(* CODESYS project LS Electric.library
   Author: Ziga Javornik
   Version: 0.0.1.1
   Description: LS Electric device libraries collection.
   Title: ZigaLibs.LsElectric
   Placeholder: ZigaLibs.LsElectric
   DefaultNamespace: ZigaLibs.LsElectric
   Company: Ziga Javornik

Project tree, tasks and I/O mapping:
  libraries: Tc2_Standard, * (Beckhoff Automation GmbH); Tc2_System, * (Beckhoff Automation GmbH); Tc3_Module, * (Beckhoff Automation GmbH); TcUnit, 1.3.1 (www.tcunit.org); ZigaLibs.Core, * (Ziga Javornik); ZigaLibs.Logging, * (Ziga Javornik)
  GVLs/
  SOURCE/
    L7NHA/
      DUTs/
        CoE/
          data type ST_L7NHA_CoE
        data type E_L7NHA_DriveState
        data type E_L7NHA_ErrorId
        data type E_L7NHA_HomingMethod
        data type E_L7NHA_ModeOfOperation
        data type ST_L7NHA_DataFromDrive
        data type ST_L7NHA_DataToDrive
        data type ST_L7NHA_DigitalInputs
        data type ST_L7NHA_EthercatData
        data type ST_L7NHA_GearRatio
        data type ST_L7NHA_HomingCommands
        data type ST_L7NHA_HomingStatus
        data type ST_L7NHA_MotionFeedback
        data type ST_L7NHA_PositioningCommands
        data type ST_L7NHA_PositioningStatus
        data type ST_L7NHA_ProfileTorqueCommands
        data type ST_L7NHA_UserUnitParams
        data type ST_L7NHA_VelocityCommands
      function block FB_L7NHA [ST]: SetGearRatio, SetHomingMethod, DisableVoltage, EnableOperation, FaultReset, Halt, Shutdown, SwitchOn, SwitchOnEnableOperation, Homing, ProfilePosition, ProfileTorque, ProfileVelocity, CalculateTorque, FB_init, GetDriveState
  TESTS/
    Test suites/
      function block FB_SUT_Tests [ST]: TestXX_Template
    program PRG_TESTS [ST]
*)

// SOURCE/L7NHA/DUTs/CoE/ST_L7NHA_CoE
TYPE ST_L7NHA_CoE :
STRUCT
	HomingMethod	: ZigaLibs_Core.ST_CoeEntry_SINT := (Index := 16#6098);
	GearRatio_Motor	: ZigaLibs_Core.ST_CoeEntry_DINT := (Index := 16#6091, Subindex := 1);
	GearRatio_Shaft	: ZigaLibs_Core.ST_CoeEntry_DINT := (Index := 16#6091, Subindex := 2);
END_STRUCT
END_TYPE

// SOURCE/L7NHA/DUTs/E_L7NHA_DriveState
{attribute 'qualified_only'}
{attribute 'strict'}
{attribute 'to_string'}
// Drive states based on the CiA402 state machine
TYPE E_L7NHA_DriveState :
(
	SWITCH_ON_DISABLED,
	READY_TO_SWITCH_ON,
	SWITCHED_ON,
	OPERATION_ENABLED,
	QUICK_STOP_ACTIVE,
	FAULT_REACTION_ACTIVE,
	FAULT
);
END_TYPE

// SOURCE/L7NHA/DUTs/E_L7NHA_ErrorId
{attribute 'qualified_only'}
{attribute 'to_string'}
// Drive error ID - same as the error displayed on the servo 7SEG display
TYPE E_L7NHA_ErrorId :
(
	NO_ERROR := 0,
	IPM_FAULT := 16#10,
	IPM_TEMPERATURE := 16#11,
	OVER_CURRENT := 16#14,
	CURRENT_OFFSET := 16#15,
	CURRENT_LIMIT_EXCEEDED := 16#16,
	CONTINIOUS_OVERLOAD := 16#21,
	DRIVE_TEMPERATURE_1 := 16#22,
	REGENERATION_OVERLOAD := 16#23,
	MOTOR_CABLE_OPEN := 16#24,
	SURROUNDING_TEMPERATURE := 16#25,
	ENCODER_TEMPERATURE := 16#26,
	ECONDER_COMMUNICATION := 16#30,
	ENCODER_CABLE_OPEN := 16#31,
	ENCODER_DATA := 16#32,
	MOTOR_SETTINGS := 16#33,
	Z_PHASE_OPEN := 16#34,
	LOW_BATTERY := 16#35,
	SINUSODIAL_ENCODER_AMPLITUDE := 16#36,
	SINUSODIAL_ENCODER_FREQUENCY := 16#37,
	ENCODER_SETTING_ERROR := 16#38,
	UNDER_VOLTAGE := 16#40,
	OVER_VOLTAGE := 16#41,
	MAIN_POWER_FAIL := 16#42,
	CONTROL_POWER_FAIL := 16#43,
	OVER_SPEED_LIMIT := 16#50,
	POS_FOLLOWING := 16#51,
	EXCESSIVE_SPEED_DEVIATION := 16#53,
	PARAMETER_CHECKSUM := 16#63,
	FACTORY_SETTING := 16#71
) UINT;
END_TYPE

// SOURCE/L7NHA/DUTs/E_L7NHA_HomingMethod
{attribute 'qualified_only'}
{attribute 'strict'}
{attribute 'to_string'}
// All the different homing methods
TYPE E_L7NHA_HomingMethod :
(
	DISABLED 									:= 0,	// Homing is disabled
	NEGATIVE_SWITCH_INDEX_REVERSE_DIRECTION 	:= 1, 	// The drive returns to the home position with the negative limit switch (NOT) and the Index (Z) pulse while driving in the reverse direction.
	POSITIVE_SWITCH_INDEX_FORWARD_DIRECTION 	:= 2, 	// The drive returns to the home position with the positive limit switch (POT) and the Index (Z) pulse while driving in the forward direction.
	HOME_SWITCH_INDEX_FORWARD_DIRECTION_7 		:= 7,	// The drive returns to the home position with the home switch (HOME) and the Index (Z) pulse while driving in the forward direction. When the positive limit switch (POT) is input during homing, the drive will switch its driving direction.
	HOME_SWITCH_INDEX_FORWARD_DIRECTION_8 		:= 8,	// The drive returns to the home position with the home switch (HOME) and the Index (Z) pulse while driving in the forward direction. When the positive limit switch (POT) is input during homing, the drive will switch its driving direction.
	HOME_SWITCH_INDEX_FORWARD_DIRECTION_9 		:= 9,	// The drive returns to the home position with the home switch (HOME) and the Index (Z) pulse while driving in the forward direction. When the positive limit switch (POT) is input during homing, the drive will switch its driving direction.
	HOME_SWITCH_INDEX_FORWARD_DIRECTION_10 		:= 10,	// The drive returns to the home position with the home switch (HOME) and the Index (Z) pulse while driving in the forward direction. When the positive limit switch (POT) is input during homing, the drive will switch its driving direction.
	HOME_SWITCH_INDEX_REVERSE_DIRECTION_11 		:= 11,	// The drive returns to the home position with the home switch (HOME) and the Index (Z) pulse while driving in the reverse direction. When the negative limit switch (NOT) is input during homing, the drive will switch its driving direction.
	HOME_SWITCH_INDEX_REVERSE_DIRECTION_12 		:= 12,	// The drive returns to the home position with the home switch (HOME) and the Index (Z) pulse while driving in the reverse direction. When the negative limit switch (NOT) is input during homing, the drive will switch its driving direction.
	HOME_SWITCH_INDEX_REVERSE_DIRECTION_13 		:= 13,	// The drive returns to the home position with the home switch (HOME) and the Index (Z) pulse while driving in the reverse direction. When the negative limit switch (NOT) is input during homing, the drive will switch its driving direction.
	HOME_SWITCH_INDEX_REVERSE_DIRECTION_14 		:= 14,	// The drive returns to the home position with the home switch (HOME) and the Index (Z) pulse while driving in the reverse direction. When the negative limit switch (NOT) is input during homing, the drive will switch its driving direction.
	HOME_SWITCH_FORWARD_DIRECTION 				:= 24,	// The drive returns to the home position with the home switch (HOME) while driving in the forward direction. When the positive limit switch (POT) is input during homing, the drive will switch its driving direction.
	HOME_SWITCH_REVERSE_DIRECTION 				:= 28,	// The drive returns to the home position with the home switch (HOME) while driving in the reverse direction. When the negative limit switch (NOT) is input during homing, the drive will switch its driving direction.
	INDEX_REVERSE_DIRECTION 					:= 33,	// The drive returns to the home position with the Index (Z) pulse while driving in the reverse direction.
	INDEX_FORWARD_DIRECTION 					:= 34,	// The drive returns to the home position with the Index (Z) pulse while driving in the forward direction.
	TO_THE_CURRENT_POSITION 					:= 35,	// Sets the current position as the origin.
	NEGATIVE_STOPPER_INDEX_REVERSE_DURECTION	:= -1,	// The drive returns to the home position with the negative stopper and the Index (Z) pulse while driving in the reverse direction.
	POSITIVE_STOPPER_INDEX_FORWARD_DIRECTION 	:= -2,	// The drive returns to the home position with the positive stopper and the Index (Z) pulse while driving in the forward direction.
	REVERSE_STOPPER_REVERSE_DIRECTION 			:= -3,	// The drive returns to the home position with the negative stopper while driving in the reverse direction.
	POSITIVE_STOPPER_FORWARD_DIRECTION 			:= -4	// The drive returns to the home position with the positive stopper while driving in the forward direction.
) SINT;
END_TYPE

// SOURCE/L7NHA/DUTs/E_L7NHA_ModeOfOperation
{attribute 'qualified_only'}
{attribute 'to_string'}
// All the possible drive modes
TYPE E_L7NHA_ModeOfOperation :
(
	PROFILE_POSITION 		:= 1,
	PROFILE_VELOCITY 		:= 3,
	PROFILE_TORQUE 			:= 4,
	HOMING					:= 6,
	INTERPOLATED_POSITION	:= 7,
	CYCLIC_SYNC_POSITION	:= 8,
	CYCLIC_SYNC_VELOCITY	:= 9,
	CYCLIC_SYNC_TORQUE		:= 10
)SINT;
END_TYPE

// SOURCE/L7NHA/DUTs/ST_L7NHA_DataFromDrive
TYPE ST_L7NHA_DataFromDrive :
STRUCT
	StatusWord			: WORD;		// Status word
	ModeOfOperation		: SINT;		// Actual mode of operation
	ErrorCode			: E_L7NHA_ErrorId;		// Most recent error code
	DigitalInputs		: UDINT;	// Info on various digital inputs
	MotionFeedback		: ST_L7NHA_MotionFeedback;	// Motion feedback from the drive
END_STRUCT
END_TYPE

// SOURCE/L7NHA/DUTs/ST_L7NHA_DataToDrive
TYPE ST_L7NHA_DataToDrive :
STRUCT
	// Control
	ControlWord					: WORD;	// Control word
	ModeOfOperation				: SINT;	// Mode of operation
	
	// Positioning mode
	ProfileVelocity				: DINT;	// Target velocity in PP mode
	TargetPosition				: DINT;	// Target position in PP mode
	MaximumProfileVelocity		: UDINT; // Maximum velocity in PP mode
	ProfileAcceleration			: UDINT; // Deceleration UU/s^2 when using PP mode
	ProfileDeceleration			: UDINT; // Acceleration UU/s^2 when using PP mode
	
	TorqueCommands	: ST_L7NHA_ProfileTorqueCommands;
	
	// Velocity mode
	TargetVelocity				: DINT;	// Target velocity in PV mode
END_STRUCT
END_TYPE

// SOURCE/L7NHA/DUTs/ST_L7NHA_DigitalInputs
TYPE ST_L7NHA_DigitalInputs :
STRUCT
	POT_SW		: BOOL;
	NOT_SW		: BOOL;
	HOME_SW		: BOOL;
	DI1_OPEN	: BOOL;
	DI2_OPEN	: BOOL;
	DI3_OPEN	: BOOL;
	DI4_OPEN	: BOOL;
	DI5_OPEN	: BOOL;
	DI6_OPEN	: BOOL;
	DI7_OPEN	: BOOL;
	DI8_OPEN	: BOOL;
	STO_OPEN	: BOOL;
END_STRUCT
END_TYPE

// SOURCE/L7NHA/DUTs/ST_L7NHA_EthercatData
TYPE ST_L7NHA_EthercatData :
STRUCT
	MasterNetID		: AMSNETID;
	SlaveAddress	: UINT;
END_STRUCT
END_TYPE

// SOURCE/L7NHA/DUTs/ST_L7NHA_GearRatio
TYPE ST_L7NHA_GearRatio :
STRUCT
	Motor	: DINT;
	Shaft	: DINT;
END_STRUCT
END_TYPE

// SOURCE/L7NHA/DUTs/ST_L7NHA_HomingCommands
TYPE ST_L7NHA_HomingCommands :
STRUCT
	Start							: BOOL;	// Starts homing procedure
	Enable							: BOOL;	// Homing will only be execute if this flag is set to true
	HomingMethod					: E_L7NHA_HomingMethod; // Defines homing method that will be used for the axis - bEnableCoeReadWrite needs to be set to TRUE for this parameter to be written
	Acceleration					: UDINT; // Acceleration in UU/s^2 - bEnableCoeReadWrite needs to be set to TRUE for this parameter to be written
	SpeedWhileSearchingForSwitch	: UDINT; // Speed at which homing will be moving axis when searching for the physical switch - bEnableCoeReadWrite needs to be set to TRUE for this parameter to be written
	SpeedWhileSearchingForZero		: UDINT; // Speed at which homing will be moving axis after switch has been found and axis is looking for index pulse - bEnableCoeReadWrite needs to be set to TRUE for this parameter to be written
END_STRUCT
END_TYPE

// SOURCE/L7NHA/DUTs/ST_L7NHA_HomingStatus
TYPE ST_L7NHA_HomingStatus :
STRUCT
	InProgress			: BOOL; // Homing in progress
	NotStarted			: BOOL; // Homing stopped or not started
	TargetNotReached	: BOOL; // Performed homing operation, but the not reach the target
	Completed			: BOOL; // Homing completed
	ErrorSpeedNotZero	: BOOL; // Homing error; speed not equal to 0
	ErrorSpeedIsZero	: BOOL; // Homing error; speed equal to 0
END_STRUCT
END_TYPE

// SOURCE/L7NHA/DUTs/ST_L7NHA_MotionFeedback
TYPE ST_L7NHA_MotionFeedback :
STRUCT
	TargetTorque		: INT;	// Target torque in .1 * rated torque
	ActualTorque		: INT;	// Torque .1 * rated torque
	
	TargetPosition		: DINT;	// Target position in user units
	ActualPosition		: DINT;	// Position in user units

	TargetMotorSpeed	: INT;	
	ActualMotorSpeed	: INT;	// Motor speed in RPM

	TargetVelocity		: DINT;	// Target velocity in user units
	ActualVelocity		: DINT;	// Velocity in user units
END_STRUCT
END_TYPE

// SOURCE/L7NHA/DUTs/ST_L7NHA_PositioningCommands
TYPE ST_L7NHA_PositioningCommands :
STRUCT
	VelocitySetpoint		: DINT;		// Velocity setpoint when in positioning mode
	MaxVelocity				: UDINT;	// Maximum allowed velocity when in positioning mode
	TargetPosition			: DINT;		// Target position
	GoToPosition			: BOOL;		// Positioning will be executed on rising edge
	ImmediatePositioning	: BOOL;		// If set to TRUE target position will be sent to the drive immediately and executed - otherwise the target only updates on GoToPosition call	
	EnablePositioning		: BOOL;		// Positioning will only be executed when this flag is set to true
END_STRUCT
END_TYPE

// SOURCE/L7NHA/DUTs/ST_L7NHA_PositioningStatus
TYPE ST_L7NHA_PositioningStatus :
STRUCT
	TargetPositionReached	 		: BOOL;	// TRUE if position has been reached
	SetpointAcknowledged			: BOOL;	// TRUE if new setpoint has been acknowledged
	PositionalError					: BOOL;	// TRUE if positioning error is detected
END_STRUCT
END_TYPE

// SOURCE/L7NHA/DUTs/ST_L7NHA_ProfileTorqueCommands
TYPE ST_L7NHA_ProfileTorqueCommands :
STRUCT
	TargetTorque			: UINT; // Target value - 0.1% of rated torque
	MaxTorque				: UINT; // Limits torque in both directions - 0.1% of rated torque
	MaximumProfileVelocity 	: UDINT; // Maximum velocity when driving using the torque mode - UU/s
	TorqueSlope				: UDINT; // Slope of the generated torque profile - 0.1%/s
	PositiveTorqueLimit		: UINT;	// Limit when driving in positive direction - 0.1%
	NegativeTorqueLimit		: UINT;	// Limit when driving in negative direction - 0.1%
	TorqueOffset			: UINT;	// Offset added to the TargeTorque
END_STRUCT
END_TYPE

// SOURCE/L7NHA/DUTs/ST_L7NHA_UserUnitParams
// Specifies custom user unit data that can be used for further conversion from within the block
TYPE ST_L7NHA_UserUnitParams :
STRUCT
	(* Use this to specify if you want to use custom user unit, different from the one set on the drive. 
	This can be useful if you have low user unit and want to sue higher unit inside the program since 
	scaling is done within the block for simplciyt sake. If you don't want to use actual units leave this at 1 (or 0 - internal check will ommit any calculation if set to 0).
	Example:
		- Gearbox ratio is set so that user unit is 1um.
		- You want to use milimeters as your unit inside the program.
		- Set the divisor to 1000 - UU outside the block is then 1mm = 1value, instead of 1000 = 1000um = 1mm..*)
	GearboxRatioUnitDivisor	: DINT := 1;
	
	(*User unit for velocity is by deafult in UU/s. Use this to automatically convert velocity to UU/<CustomVelocityTimeUnitDivisor>*seconds
	Example:
		- You have set up the gearbox to be in milimeters per 1 unit.
		- You want the speed to be in mm/minute instead of defautl mm/second.
		- Set this parameter to 60, this way velocity feedback will be multiplied by 60, which will return velocity in mm/min 
		  and velocity setpoint will be divided by 60 to specify the speed to the drive in UU/seconds, which is the only option.*)	
	CustomVelocityTimeUnitDivisor		: REAL := 1;
END_STRUCT
END_TYPE

// SOURCE/L7NHA/DUTs/ST_L7NHA_VelocityCommands
TYPE ST_L7NHA_VelocityCommands :
STRUCT
	VelocitySetpoint	: DINT;	// Target velocity in UU/s used in Profile Velocity mode
END_STRUCT
END_TYPE

// SOURCE/L7NHA/FB_L7NHA
FUNCTION_BLOCK FB_L7NHA EXTENDS ZigaLibs_Core.FB_HasInstanceNameAndPath

VAR_INPUT
	bEnable					: BOOL;	// Enable axis
	bReset					: BOOL;	// Reset if an eror is present
	bHalt					: BOOL; // Halts current operation - after setting this to FALSE previous operation is continuoued
	bQuickStop				: BOOL;	// Drive will execute a quick stop
	
	nAcceleration			: UDINT;	// Axis acceleration in UU/s^2
	nDeceleration			: UDINT;	// Axis deceleration in UU/s^
	
	eModeOfOperation		: E_L7NHA_ModeOfOperation;	// Mode of operation
	
	stVelocityCommands		: ST_L7NHA_VelocityCommands;		// Velocity commands when in profile velocity mode
	stPositioningCommands	: ST_L7NHA_PositioningCommands;		// Positioning commands when in profile position mode
	stHomingCommands		: ST_L7NHA_HomingCommands;			// Homing commands when in homing sequence
	stProfileTorqueCommands	: ST_L7NHA_ProfileTorqueCommands;	// Profile torque commands when using Profile Torque mode
	
	fRatedTorque			: REAL; // Rated torque in mNm - required for torque calculation

	stGearRatio				: ST_L7NHA_GearRatio;	// Used to set gear ratio
END_VAR

VAR_OUTPUT
	eAxisState			: E_L7NHA_DriveState;	// Axis state, actual state reported back from drive
	
	eErrorCode			: E_L7NHA_ErrorId;	// Error code, if drive is in fault state
	
	bHomingRequired		: BOOL;	// If homing is required, this flag will be set to true (usually after a power reset)
	
	bMovingPositive		: BOOL;	// Indicating axis is rotating in positive direction
	bMovingNegative		: BOOL;	// Indicating axis is rotating in negative direction
	
	stPositioningStatus	: ST_L7NHA_PositioningStatus;	// Status of the positioning procedure - only valid when in positioning mode
	stHomingStatus		: ST_L7NHA_HomingStatus;		// Status of the homing procedure - only valid when in homing mode
	
	fCalculatedActualTorque	: REAL;
	fCalculatedTargetTorque	: REAL;
	
	eActualModeOfOperation	: E_L7NHA_ModeOfOperation;
	stMotionFeedback		: ST_L7NHA_MotionFeedback;	// Motion feedback from the drive

	stDigitalInputs	:		 ST_L7NHA_DigitalInputs;
	
	bModeOfOperationNotImplemented	: BOOL;	// Will be TRUE if the selected mode of operation is not implemented (axis has to be in enabled state for this flag to be valid!)
END_VAR

// Local variables
VAR
	eAxisStateInternal					: E_L7NHA_DriveState;
	stDataToDriveInternal				: ST_L7NHA_DataToDrive;
	TonCommandTimeout					: Tc2_Standard.TON := (PT := T#1S);
	RtrigMoveToPosition					: Tc2_Standard.R_TRIG;
	RtrigStartHoming					: Tc2_Standard.R_TRIG;
	nPreviousPosition					: DINT;
	RtrigResetTrigger					: Tc2_Standard.R_TRIG;
	RtrigHomingFinished					: Tc2_Standard.R_TRIG;
	TonMotorMovingStatusValid			: Tc2_Standard.TON;
	RtrigModeOfOperationNotImplemented	: Tc2_Standard.R_TRIG;
	eModeOfOpereationOld				: E_L7NHA_ModeOfOperation;
	_logger								: REFERENCE TO ZigaLibs_Logging.I_Logger;
	_sb									: ZigaLibs_Core.FB_StringBuilder;
	_coeEntries							: ST_L7NHA_CoE;
END_VAR

// IO
VAR
	stDataFromDrive	AT %I* : ST_L7NHA_DataFromDrive;
	stDataToDrive	AT %Q* : ST_L7NHA_DataToDrive;
	stAmsAddress	AT %I* : Global.AMSADDR;
END_VAR

// Sometimes axis wont go to enabled - in that case a timeout should be triggered
TonCommandTimeout(in := eAxisStateInternal = E_L7NHA_DriveState.OPERATION_ENABLED);
// Reset triggering
RtrigResetTrigger(CLK := bReset);


// Abs encoder value is not valid if bit 14 is FALSE (homing has not been completed yet after a power reset/encoder error)
bHomingRequired := stDataFromDrive.StatusWord.14 = FALSE;

// Calling halt will overwrite this - to enable automatic clearing, setting it to false by default
stDataToDriveInternal.ControlWord.8 := FALSE;

// State machine based on the drive's feedback
eAxisStateInternal := THIS^.GetDriveState();

bModeOfOperationNotImplemented := FALSE;
		
// State machine based on actual state reported back from the drive
CASE eAxisStateInternal OF
	E_L7NHA_DriveState.SWITCH_ON_DISABLED:	
		IF bEnable THEN
			Shutdown();
		ELSE
			DisableVoltage();
		END_IF
	
	E_L7NHA_DriveState.READY_TO_SWITCH_ON:
		IF NOT TonCommandTimeout.Q THEN
			SwitchOnEnableOperation();
		END_IF
		
	E_L7NHA_DriveState.OPERATION_ENABLED:
		TonCommandTimeout.IN := FALSE;
		SwitchOnEnableOperation();

		// Execute different mode based on mode of operation setting
		CASE eModeOfOperation OF
			E_L7NHA_ModeOfOperation.PROFILE_POSITION:
				ProfilePosition();
				
			E_L7NHA_ModeOfOperation.PROFILE_VELOCITY:
				ProfileVelocity();
				
			E_L7NHA_ModeOfOperation.HOMING:
				Homing();
				
			E_L7NHA_ModeOfOperation.PROFILE_TORQUE:
				ProfileTorque();
				
			ELSE
				bModeOfOperationNotImplemented := TRUE;
				IF eModeOfOperation <> eModeOfOpereationOld THEN
					IF __ISVALIDREF(_logger) THEN
						_logger.LogError(_sb.Reset()
							.AddString('L7NHA axis ')
							.AddWithDblQuotationMarks(THIS^.InstanceName)
							.AddString(': Mode of operation is not supported! Selected mode is ')
							.AddWithDblQuotationMarks(TO_STRING(eModeOfOperation))
							.Create());
					END_IF
				END_IF
		END_CASE
		
	E_L7NHA_DriveState.FAULT:
		IF RtrigResetTrigger.Q THEN
			FaultReset();
		ELSE
			stDataToDriveInternal.ControlWord.7 := FALSE;
		END_IF

END_CASE

// Override any command if enable is false (transitioning states) - exception is fault, where reset needs to be sent
IF NOT bEnable AND eAxisStateInternal <> E_L7NHA_DriveState.FAULT THEN
	DisableVoltage();
END_IF

// Halt - has a different meaning in PP,PV or homing 
// Usally it "pauses" the current procedure and after halt is set to FALSE drive will proceed where it left off
IF bHalt THEN
	Halt();
END_IF

// Quick stop
IF bQuickStop THEN
	stDataToDriveInternal.ControlWord.1 := bQuickStop;
	stDataToDriveInternal.ControlWord.2 := NOT bQuickStop;
END_IF

// Setting acceleration/deceleration always
stDataToDriveInternal.ProfileAcceleration := nAcceleration;
stDataToDriveInternal.ProfileDeceleration := nDeceleration;

// Mode of operation
stDataToDriveInternal.ModeOfOperation := eModeOfOperation;


// =======================================================================
// ==================== SETTING FB OUTPUTS ===============================
// =======================================================================

// Axis state
eAxisState := eAxisStateInternal;

// Overwriting status for positioning/homing if not in that mode
// Clear homing status if not in that mode
IF eModeOfOperation <> E_L7NHA_ModeOfOperation.HOMING THEN
	MEMSET(
		destAddr := ADR(stHomingStatus),
		n := SIZEOF(stHomingStatus),
		fillByte := 0);
END_IF
 
// Clear positioning status if not in that mode
IF eModeOfOperation <> E_L7NHA_ModeOfOperation.PROFILE_POSITION THEN
	MEMSET(
		destAddr := ADR(stPositioningStatus),
		n := SIZEOF(stPositioningStatus),
		fillByte := 0);
END_IF

// Motion status
TonMotorMovingStatusValid(
	IN := nPreviousPosition <> stDataFromDrive.MotionFeedback.ActualPosition,
	PT := T#30MS);

bMovingPositive := (nPreviousPosition < stDataFromDrive.MotionFeedback.ActualPosition) AND TonMotorMovingStatusValid.Q;
bMovingNegative := (nPreviousPosition > stDataFromDrive.MotionFeedback.ActualPosition) AND TonMotorMovingStatusValid.Q;
nPreviousPosition := stDataFromDrive.MotionFeedback.ActualPosition;

// Digital inputs mapping
stDigitalInputs.NOT_SW := stDataFromDrive.DigitalInputs.0;
stDigitalInputs.POT_SW := stDataFromDrive.DigitalInputs.1;
stDigitalInputs.DI1_OPEN := stDataFromDrive.DigitalInputs.16;
stDigitalInputs.DI2_OPEN := stDataFromDrive.DigitalInputs.17;
stDigitalInputs.DI3_OPEN := stDataFromDrive.DigitalInputs.18;
stDigitalInputs.DI4_OPEN := stDataFromDrive.DigitalInputs.19;
stDigitalInputs.DI5_OPEN := stDataFromDrive.DigitalInputs.20;
stDigitalInputs.DI6_OPEN := stDataFromDrive.DigitalInputs.21;
stDigitalInputs.DI7_OPEN := stDataFromDrive.DigitalInputs.22;
stDigitalInputs.DI8_OPEN := stDataFromDrive.DigitalInputs.23;
stDigitalInputs.STO_OPEN := stDataFromDrive.DigitalInputs.31;

// Error code
IF eErrorCode <> stDataFromDrive.ErrorCode THEN
	IF __ISVALIDREF(_logger) THEN
		IF stDataFromDrive.ErrorCode = E_L7NHA_ErrorId.NO_ERROR THEN
			_logger.LogInfo(_sb.Reset()
				.AddString('L7NHA axis ')
				.AddWithDblQuotationMarks(THIS^.InstanceName)
				.AddString(' error no longer active.')
				.Create());
		ELSE
			_logger.LogError(_sb.Reset()
				.AddString('L7NHA axis ')
				.AddWithDblQuotationMarks(THIS^.InstanceName)
				.AddString(' error active! Error code: ')
				.AddString(TO_STRING(stDataFromDrive.ErrorCode))
				.AddString(' !')
				.Create());
		END_IF
	END_IF
END_IF

eErrorCode := stDataFromDrive.ErrorCode;

// Motion feedback from drive
stMotionFeedback := stDataFromDrive.MotionFeedback;
// Convert position/velocity to custom units

stMotionFeedback := stDataFromDrive.MotionFeedback;

fCalculatedActualTorque := CalculateTorque(fRatedTorque := fRatedTorque, nDriveTorqueFeedback := stDataFromDrive.MotionFeedback.ActualTorque);
fCalculatedTargetTorque := CalculateTorque(fRatedTorque := fRatedTorque, nDriveTorqueFeedback := stDataFromDrive.MotionFeedback.TargetTorque);

// Actual mode of operation, read from the drive
eActualModeOfOperation := stDataFromDrive.ModeOfOperation;

eModeOfOpereationOld := eModeOfOperation;

// =======================================================================
// ==================== SETTING OUTPUT STRUCTURE TO DRIVE ================
// =======================================================================
stDataToDrive := stDataToDriveInternal;

// Observes the stGearRatio.Shaft and stGearRatio.Motor. If the setting changes the new value is written to the CoE parameter.
METHOD pubLIC SetGearRatio : BOOL

VAR_INST
	coeReadWrite	: ZigaLibs_Core.FB_CoeReadWrite;
	sb				: ZigaLibs_Core.FB_StringBuilder;
	writeShaftDone 	: BOOL;
	writeMotorDone	: BOOL;
END_VAR
IF writeMotorDone = FALSE THEN
	IF coeReadWrite.WriteAny(
		Value := stGearRatio.Motor, 
		CoeEntry := ADR(_coeEntries.GearRatio_Motor), 
		SlaveAddr := stAmsAddress)
	THEN
		writeMotorDone := TRUE;
		IF __ISVALIDREF(_logger) then
			sb.Reset()
				.AddString('L7NHA axis ')
				.AddWithDblQuotationMarks(THIS^.InstanceName)
				.AddString(': Motor gear ratio changed to ')
				.AddString(TO_STRING(stGearRatio.Motor));
			_logger.LogInfo(sb.Create());
		END_IF
	END_IF	
END_IF

IF writeMotorDone THEN
	IF coeReadWrite.WriteAny(
		Value := stGearRatio.Shaft, 
		CoeEntry := ADR(_coeEntries.GearRatio_Motor), 
		SlaveAddr := stAmsAddress)
	THEN
		SetGearRatio := TRUE;
		writeMotorDone := FALSE;
		IF __ISVALIDREF(_logger) then
			sb.Reset()
				.AddString('L7NHA axis ')
				.AddWithDblQuotationMarks(THIS^.InstanceName)
				.AddString(': Shaft gear ratio changed to ')
				.AddString(TO_STRING(stGearRatio.Shaft));
			_logger.LogInfo(sb.Create());
		END_IF
	END_IF		
END_IF
END_METHOD

// Writes the current homing method provided in stHomingCommands.HomingMethod to the CoE of the axis. Returns TRUE when done
METHOD PUBLIC SetHomingMethod : BOOL
VAR_INST
	coeReadWrite	: ZigaLibs_Core.FB_CoeReadWrite;
	sb				: ZigaLibs_Core.FB_StringBuilder;
END_VAR
IF coeReadWrite.WriteAny(
		Value := stHomingCommands.HomingMethod, 
		CoeEntry := ADR(_coeEntries.HomingMethod), 
		SlaveAddr := stAmsAddress)
THEN 
	IF __ISVALIDREF(_logger) then
		sb.Reset()
			.AddString('L7NHA axis ')
			.AddWithDblQuotationMarks(THIS^.InstanceName)
			.AddString(': Homing method changing to ')
			.AddString(TO_STRING(stHomingCommands.HomingMethod));
		_logger.LogInfo(sb.Create());
	END_IF
	SetHomingMethod := TRUE;
END_IF
END_METHOD

METHOD PRIVATE DisableVoltage
stDataToDriveInternal.controlWord := 0;
END_METHOD

METHOD PRIVATE EnableOperation
stDataToDriveInternal.controlWord.0 := 0;
stDataToDriveInternal.controlWord.1 := 1;
stDataToDriveInternal.controlWord.2 := 1;
stDataToDriveInternal.controlWord.3 := 0;
stDataToDriveInternal.controlWord.4 := 0;
stDataToDriveInternal.controlWord.5 := 0;
stDataToDriveInternal.controlWord.6 := 0;
stDataToDriveInternal.controlWord.7 := 0;
END_METHOD

METHOD PRIVATE FaultReset
IF stDataToDriveInternal.controlWord.7 = 0 THEN
	stDataToDriveInternal.controlWord.7 := 1;
	stDataToDriveInternal.controlWord.0 := 0;
	stDataToDriveInternal.controlWord.1 := 0;
	stDataToDriveInternal.controlWord.2 := 0;
	stDataToDriveInternal.controlWord.3 := 0;
END_IF
END_METHOD

// Halts the axis for as long as called
METHOD PRIVATE Halt : BOOL
VAR_INPUT
END_VAR
stDataToDriveInternal.ControlWord.8 := TRUE;
END_METHOD

METHOD PRIVATE Shutdown
stDataToDriveInternal.controlWord.0 := 0;
stDataToDriveInternal.controlWord.1 := 1;
stDataToDriveInternal.controlWord.2 := 1;
stDataToDriveInternal.controlWord.7 := 0;
END_METHOD

METHOD PRIVATE SwitchOn
stDataToDriveInternal.controlWord.0 := 1;
stDataToDriveInternal.controlWord.1 := 1;
stDataToDriveInternal.controlWord.2 := 1;
stDataToDriveInternal.controlWord.3 := 0;
END_METHOD

METHOD PRIVATE SwitchOnEnableOperation
stDataToDriveInternal.controlWord.0 := 1;
stDataToDriveInternal.controlWord.1 := 1;
stDataToDriveInternal.controlWord.2 := 1;
stDataToDriveInternal.controlWord.3 := 1;
END_METHOD

ACTION Homing:
// Set the status of homing

// Hooming is in progress
stHomingStatus.InProgress := 
stDataFromDrive.StatusWord.10 = FALSE AND
stDataFromDrive.StatusWord.12 = FALSE AND
stDataFromDrive.StatusWord.13 = FALSE;

// Homing is not started
stHomingStatus.NotStarted := 
stDataFromDrive.StatusWord.10 = TRUE AND
stDataFromDrive.StatusWord.12 = FALSE AND
stDataFromDrive.StatusWord.13 = FALSE;	

// Target not reached	
stHomingStatus.TargetNotReached := 
stDataFromDrive.StatusWord.10 = FALSE AND
stDataFromDrive.StatusWord.12 = TRUE AND
stDataFromDrive.StatusWord.13 = FALSE;

// Homing completed
stHomingStatus.Completed := 
stDataFromDrive.StatusWord.10 = TRUE AND
stDataFromDrive.StatusWord.12 = TRUE AND
stDataFromDrive.StatusWord.13 = FALSE;

// Error - speed is not zero ????
stHomingStatus.ErrorSpeedNotZero := 
stDataFromDrive.StatusWord.10 = FALSE AND
stDataFromDrive.StatusWord.12 = FALSE AND
stDataFromDrive.StatusWord.13 = TRUE;

// Error - speed is zero ????
stHomingStatus.ErrorSpeedIsZero := 
stDataFromDrive.StatusWord.10 = TRUE AND
stDataFromDrive.StatusWord.12 = FALSE AND
stDataFromDrive.StatusWord.13 = TRUE;


RtrigStartHoming(CLK := stHomingCommands.Start);	
IF stHomingCommands.Enable = FALSE THEN
	stDataToDriveInternal.ControlWord.4 := FALSE;
ELSIF RtrigStartHoming.Q THEN
	stDataToDriveInternal.ControlWord.4 := TRUE;
END_IF

RtrigHomingFinished(CLK := stHomingStatus.Completed);
IF RtrigHomingFinished.Q THEN
	stDataToDriveInternal.ControlWord.4 := FALSE;
END_IF
END_ACTION

ACTION ProfilePosition:
// Positioning is only allowed if homing has been executed
IF NOT bHomingRequired THEN					
	// Set maximum velocity
	stDataToDriveInternal.MaximumProfileVelocity := stPositioningCommands.MaxVelocity;
	
	// Update target immediately - bit 5 is TRUE
	stDataToDriveInternal.ControlWord.5 := TRUE;
	
	// Trigger immediate update of setpoint by toggling the bit
	IF stPositioningCommands.EnablePositioning THEN
		// Toggling of bit 4 will execute the changes as soon as they are written
		IF stPositioningCommands.ImmediatePositioning THEN
			stDataToDriveInternal.ControlWord.4 := NOT stDataToDriveInternal.ControlWord.4;
			stDataToDriveInternal.ProfileVelocity := stPositioningCommands.VelocitySetpoint;
			stDataToDriveInternal.TargetPosition := stPositioningCommands.TargetPosition;
		ELSE
			// Bit 4 is only set for 1 cycle when requested by the GoToPosition trigger
			stDataToDriveInternal.ControlWord.4 := FALSE;
			// Sending values only on triger of GoToPosition property
			RtrigMoveToPosition(CLK := stPositioningCommands.GoToPosition);
			IF RtrigMoveToPosition.Q THEN
				stDataToDriveInternal.ControlWord.4 := TRUE;
				stDataToDriveInternal.ProfileVelocity := stPositioningCommands.VelocitySetpoint;
				stDataToDriveInternal.TargetPosition := stPositioningCommands.TargetPosition;
			END_IF
		END_IF
	ELSE
		Halt();
	END_IF
	
	// Positioning status from drive
	stPositioningStatus.TargetPositionReached := stDataFromDrive.StatusWord.10;
	stPositioningStatus.SetpointAcknowledged := stDataFromDrive.StatusWord.12;
	stPositioningStatus.PositionalError := stDataFromDrive.StatusWord.13;
ELSE
	// If homing has not been executed, halt axis
	Halt();
END_IF
END_ACTION

ACTION ProfileTorque:
stDataToDriveInternal.TorqueCommands := stProfileTorqueCommands;
END_ACTION

ACTION ProfileVelocity:
// Velocity mode is very simple - just send out the speed setpoint
stDataToDriveInternal.TargetVelocity := stVelocityCommands.VelocitySetpoint;
END_ACTION

METHOD PRIVATE CalculateTorque : REAL
VAR_INPUT
	fRatedTorque 			: REAL; // Rated torque in mNm
	nDriveTorqueFeedback 	: INT;	// Drives feedback (0.1% increments, -100%...+100%)
END_VAR
CalculateTorque := fRatedTorque * TO_REAL(nDriveTorqueFeedback);
END_METHOD

METHOD FB_init : BOOL
VAR_INPUT
	bInitRetains : BOOL; // if TRUE, the retain variables are initialized (warm start / cold start)
	bInCopyCode : BOOL;  // if TRUE, the instance afterwards gets moved into the copy code (online change)
	logger		: REFERENCE TO ZigaLibs_Logging.I_Logger; // If you do not want logging, simply set this variable to 0, internal checks will ommit any logging.		
END_VAR
_logger REF= logger;
END_METHOD

// Converts status word to a readable drive state enum
METHOD PRIVATE GetDriveState : E_L7NHA_DriveState
//================ SWITCH_ON_DISABLED =====================
IF stDataFromDrive.StatusWord.0 = FALSE AND
    stDataFromDrive.StatusWord.1 = FALSE AND
    stDataFromDrive.StatusWord.2 = FALSE AND
    stDataFromDrive.StatusWord.3 = FALSE AND
    stDataFromDrive.StatusWord.5 = TRUE AND 
    stDataFromDrive.StatusWord.6 = TRUE
THEN
	GetDriveState := E_L7NHA_DriveState.SWITCH_ON_DISABLED;

//================ READY_TO_SWITCH_ON =====================	
ELSIF stDataFromDrive.StatusWord.0 = TRUE AND
   	   stDataFromDrive.StatusWord.1 = FALSE AND
       stDataFromDrive.StatusWord.2 = FALSE AND
       stDataFromDrive.StatusWord.3 = FALSE AND
       stDataFromDrive.StatusWord.5 = TRUE AND 
       stDataFromDrive.StatusWord.6 = FALSE
THEN
	GetDriveState := E_L7NHA_DriveState.READY_TO_SWITCH_ON;	

//================ SWITCHED_ON ==========================	
ELSIF stDataFromDrive.StatusWord.0 = TRUE AND
   	   stDataFromDrive.StatusWord.1 = TRUE AND
       stDataFromDrive.StatusWord.2 = FALSE AND
       stDataFromDrive.StatusWord.3 = FALSE AND
       stDataFromDrive.StatusWord.5 = TRUE AND 
       stDataFromDrive.StatusWord.6 = FALSE
THEN
	GetDriveState := E_L7NHA_DriveState.SWITCHED_ON;

//================ OPERATION_ENABLED =====================	
ELSIF stDataFromDrive.StatusWord.0 = TRUE AND
   	   stDataFromDrive.StatusWord.1 = TRUE AND
       stDataFromDrive.StatusWord.2 = TRUE AND
       stDataFromDrive.StatusWord.3 = FALSE AND
       stDataFromDrive.StatusWord.5 = TRUE AND 
       stDataFromDrive.StatusWord.6 = FALSE
THEN
	GetDriveState := E_L7NHA_DriveState.OPERATION_ENABLED;

//================ FAULT_REACTION_ACTIVE =====================		
ELSIF stDataFromDrive.StatusWord.0 = TRUE AND
   	   stDataFromDrive.StatusWord.1 = TRUE AND
       stDataFromDrive.StatusWord.2 = TRUE AND
       stDataFromDrive.StatusWord.3 = TRUE AND
       stDataFromDrive.StatusWord.5 = TRUE AND 
       stDataFromDrive.StatusWord.6 = FALSE
THEN
	GetDriveState := E_L7NHA_DriveState.FAULT_REACTION_ACTIVE;

//================ FAULT =====================	
ELSIF  stDataFromDrive.StatusWord.0 = FALSE AND
   	   stDataFromDrive.StatusWord.1 = FALSE AND
       stDataFromDrive.StatusWord.2 = FALSE AND
       stDataFromDrive.StatusWord.3 = TRUE AND 
       stDataFromDrive.StatusWord.6 = FALSE
THEN
	GetDriveState := E_L7NHA_DriveState.FAULT;				
END_IF
END_METHOD

END_FUNCTION_BLOCK

// TESTS/Test suites/FB_SUT_Tests
// Subject under test
FUNCTION_BLOCK FB_SUT_Tests EXTENDS FB_TestSuite

// Create instance variables that will be accesible for all tests
VAR
END_VAR

// Call your test methods here
TestXX_Template();

METHOD PRIVATE TestXX_Template

(* Instanced variables are VERY useful for writing tests since tests are run in paralel (by default).
By instantiating local variables that are not placed on the same stack as method (values are retained between calls)
you make sure that the SUT is not changed by some other test. *)
VAR_INST
	
END_VAR

// Place temporary variables here
VAR
	
END_VAR
// The name of the test, is the same as method name!
// Use this for paralel unit tests
// TcUnit.TEST('TestXX_Template');

// Use this for running tests in sequence
IF TcUnit.TEST_ORDERED('TestXX_Template') THEN
	// Do your assertions here...
	AssertTrue(
		Condition := FALSE, 
		Message := 'Implement tests!');

	TcUnit.TEST_FINISHED();
END_IF
END_METHOD

END_FUNCTION_BLOCK

// TESTS/PRG_TESTS
PROGRAM PRG_TESTS

(* Instantiate test suites here. Naming convention for tests should be a suffix with _Tests.
Good practice for creating test methods is to end them with _test as well. *)
VAR
	fbSUT_Tests	: FB_SUT_Tests;
END_VAR

// Run tests in parallel
//TcUnit.RUN();

// Run tests in sequence, one after the other.
TcUnit.RUN_IN_SEQUENCE();

END_PROGRAM
